PROGRAM StDrool
VAR
	CaseCool: INT;
	YellowMinions: INT;
	WorkAtUS: INT;
	JustinAndAlex: INT;
	lookFly: INT;
END_VAR

CASE CaseCool OF 
	0:
		YellowMinions := WorkAtUS;
		
	1: 
		//free cars for everybody
		
	2: 
		JustinAndAlex := lookFly;
		
		
END_CASE

END_PROGRAM

(* stored: Version 1.1.0.1, ProductVersion 3.1.4024.12
   POU StDrool: Id {9af66e64-35ca-4a5c-a114-7dd5c387482a}, SpecialFunc None *)
